// TwinCAT 3 PLC project DatabasePyAds
// ProgramVersion: 3.1.4023.0
// libraries:
//   Tc2_Standard, * (Beckhoff Automation GmbH)
//   Tc2_System, * (Beckhoff Automation GmbH)
//   Tc3_Module, * (Beckhoff Automation GmbH)
// project tree:
//   / PlcTask.TcTTO
//   POUs/DatabasePyAds/ DatabasePyAds.TcPOU, E_LogType.TcDUT, ST_Config.TcDUT, ST_LogData.TcDUT, ST_PyAdsConfig.TcDUT, ST_PyAdsQuit.TcDUT
//   POUs/ MAIN.TcPOU

CONFIGURATION DatabasePyAds
    RESOURCE PLC ON TwinCAT3
        TASK PlcTask(INTERVAL := T#10ms, PRIORITY := 20);
        PROGRAM MAIN WITH PlcTask : MAIN;
    END_RESOURCE
END_CONFIGURATION

// ---- POUs/DatabasePyAds/E_LogType.TcDUT
{attribute 'qualified_only'}
TYPE E_LogType:
(
	Info := 1, 
	Warnung := 2, 
	Fehler := 3
) BYTE;
END_TYPE

// ---- POUs/DatabasePyAds/ST_Config.TcDUT
TYPE ST_Config:
  STRUCT
    sLocalAmsNetId: T_AmsNetId;
    sMachineName  : STRING(20) := 'L123';
    nMachineId    : UINT       := 999;
    sPlcIP        : T_IPv4Addr;
    sLanguage     : STRING(20) := 'default';
  END_STRUCT
END_TYPE

// ---- POUs/DatabasePyAds/ST_LogData.TcDUT
TYPE ST_LogData:
  STRUCT
    bExecute: BOOL;
    sMsg    : STRING(MAX_STRING_LENGTH);
    sStation: STRING(20);
    nUserId : UDINT;
    eLogType: E_LogType;
  END_STRUCT
END_TYPE

// ---- POUs/DatabasePyAds/ST_PyAdsConfig.TcDUT
TYPE ST_PyAdsConfig :
STRUCT
	sDatabase: STRING;
	sTypeDatabase: STRING;
	sHost: STRING;
	sUser: STRING;
	sPassword: STRING;
END_STRUCT
END_TYPE

// ---- POUs/DatabasePyAds/ST_PyAdsQuit.TcDUT
TYPE ST_PyAdsQuit:
  STRUCT
    bDone : BOOL;
    bError: BOOL;
  END_STRUCT
END_TYPE

// ---- POUs/MAIN.TcPOU
PROGRAM MAIN
VAR
END_VAR

DatabasePyAds();

END_PROGRAM

// ---- POUs/DatabasePyAds/DatabasePyAds.TcPOU
PROGRAM DatabasePyAds
VAR_INPUT
  bGetTest: BOOL;
  stLog  : ST_LogData;
END_VAR
VAR_OUTPUT
  stGetTestQuit: ST_PyAdsQuit;
  stLogQuit: ST_PyAdsQuit;  
END_VAR
VAR
  bExecute: BOOL;
  bDone   : BOOL;
  bBusy   : BOOL;
  bError  : BOOL;
  stConfig: ST_PyAdsConfig;

  diRows       : DINT;
  diColumns    : DINT;
  saRequest    : ARRAY[1..cUBoundRequestArray] OF STRING(cMaxStringLength);
  saColumnsName: ARRAY[1..cMaxColumns] OF STRING(cStringLength);
  saTableValues: ARRAY[1..cMaxRows, 1..cMaxColumns] OF STRING(cMaxStringLength);
  sError       : STRING(cMaxStringLength);
  sVersion     : STRING(cStringLength);

  tonTimeout       : TON := (PT := T#60S);
  nState, nSubState: INT;
  i                : INT;
  _iReq            : INT;
  iStateBranch     : INT;
    bWithAnswer : BOOL;
  
END_VAR

VAR CONSTANT
  cMaxRows           : UDINT := 200;
  cMaxColumns        : UDINT := 30;
  cStringLength      : UDINT := 80;
  cMaxStringLength   : UDINT := MAX_STRING_LENGTH;
  cUBoundRequestArray: UDINT := 20;

  // Databases
  stDbMySql: ST_PyAdsConfig := (sDatabase := 'test',
    sTypeDatabase                         := 'mysql',
    sHost                                 := '192.168.1.7',
    sUser                                 := 'test',
    sPassword                             := 'test');
  stDbMySql2: ST_PyAdsConfig := (sDatabase := 'test2',
    sTypeDatabase                          := 'mysql',
    sHost                                  := '192.168.1.7',
    sUser                                  := 'test',
    sPassword                              := 'test');
  stDbMssql: ST_PyAdsConfig := (sDatabase := 'test',
    sTypeDatabase                         := 'mssql',
    sHost                                 := '192.168.1.250',
    sUser                                 := 'test',
    sPassword                             := 'test');

  cReset  : INT := 0;
  cInitial: INT := 1;
  cTest   : INT := 10;
  cLog    : INT := 100;
END_VAR

CASE nState OF
  cReset:
    stConfig := stDbMssql; (* default database *)
    nState   := cInitial;

  cInitial:
    IF bBusy THEN
      ;
    ELSIF bGetTest THEN
      nState := cTest;
    ELSIF stLog.bExecute THEN
      stConfig := stDbMySql2;
      nState   := cLog;
    END_IF

    IF nState > cInitial THEN
      tonTimeout(IN := FALSE);
      nSubState := 0;
      bDone     := FALSE;
      bError    := FALSE;
      // clean strings
      MEMSET(ADR(saRequest), 0, SIZEOF(saRequest));
      MEMSET(ADR(saColumnsName), 0, SIZEOF(saColumnsName));
      MEMSET(ADR(saTableValues), 0, SIZEOF(saTableValues));
      MEMSET(ADR(sError), 0, SIZEOF(sError));
    END_IF

  cTest:
    stGetTestQuit := GetTest(bRunQuery := bGetTest);
  cLog:
    stLogQuit := SetLog(stRunQuery := stLog);

END_CASE;

METHOD PRIVATE _ResetStates
nState := cReset;
nSubState := cReset;
END_METHOD

METHOD PRIVATE _Timeout: BOOL
IF tonTimeout.Q THEN
	_ResetStates();
	bError := TRUE;
	bExecute := FALSE;
END_IF
IF NOT bBusy THEN
	tonTimeout(IN := TRUE);
END_IF
END_METHOD

METHOD PRIVATE GetTest: ST_PyAdsQuit
VAR_IN_OUT
	bRunQuery: BOOL;
END_VAR
CASE nSubState OF
0:
	iReq := 1;
	saRequest[iReq] := 'SELECT leit_set_log';
	saRequest[iReq] := ' (';
	saRequest[iReq] := '1';
	saRequest[iReq] := ',';
	saRequest[iReq] := INT_TO_STRING(stLog.eLogType);
	saRequest[iReq] := ',"';
	saRequest[iReq] := stLog.sStation;
	saRequest[iReq] := '","';
	saRequest[iReq] := stLog.sMsg;
	saRequest[iReq] := '")';

	bWithAnswer := TRUE;
	bExecute := TRUE;
	nSubState := nSubState + 1;
1:
	IF NOT bExecute THEN
		nSubState := nSubState + 1;
	END_IF
2:
	IF bDone OR bError THEN
		IF bError THEN
      FOR i := 1 TO DINT_TO_INT(diRows) DO
				// log
			END_FOR
		END_IF		
		bRunQuery := FALSE;
		_ResetStates();
	END_IF
END_CASE

IF _Timeout() THEN
	bRunQuery := FALSE;
END_IF
END_METHOD

{attribute ‘monitoring’:=’variable’}
PROPERTY iReq : INT
GET
VAR
  _iReq: INT;
END_VAR
iReq := _iReq;
_iReq := iReq + 1;
END_GET
SET
_iReq := iReq;
END_SET
END_PROPERTY

METHOD PRIVATE SetLog: ST_PyAdsQuit
VAR_IN_OUT
	stRunQuery: ST_LogData;
END_VAR
CASE nSubState OF
0:
	iReq := 1;
	saRequest[iReq] := 'SELECT leit_set_log';
	saRequest[iReq] := ' (';
	saRequest[iReq] := '1';
	saRequest[iReq] := ',';
	saRequest[iReq] := INT_TO_STRING(stRunQuery.eLogType);
	saRequest[iReq] := ',"';
	saRequest[iReq] := stRunQuery.sStation;
	saRequest[iReq] := '","';
	saRequest[iReq] := stRunQuery.sMsg;
	saRequest[iReq] := '")';

	bWithAnswer := TRUE;
	bExecute := TRUE;
	nSubState := nSubState + 1;
1:
	IF NOT bExecute THEN
		nSubState := nSubState + 1;
	END_IF
2:
	IF bDone OR bError THEN
		IF bError THEN
      FOR i := 1 TO DINT_TO_INT(diRows) DO
				// log
			END_FOR
		END_IF		
		stRunQuery.bExecute := FALSE;
		_ResetStates();
	END_IF
END_CASE

IF _Timeout() THEN
	stRunQuery.bExecute := FALSE;
END_IF
END_METHOD

END_PROGRAM
